// TIA Portal V17 export
// export: Created 2024-08-26T21:07:17.5555662Z, ExportSetting WithDefaults, DisplayName Totally Integrated Automation Portal, DisplayVersion V17 Update 7, DisplayName TIA Portal Openness, DisplayVersion V17 Update 7, DisplayName TIA Portal Version Control Interface, DisplayVersion V17, DisplayName SINAMICS Startdrive Advanced, DisplayVersion V17 SP2, DisplayName SINAMICS Startdrive G110M, G120, G120C, G120D, G120P, G115D, DisplayVersion V17 SP2, DisplayName SINAMICS Startdrive G130, G150, S120, S150, SINAMICS MV, S210, DisplayVersion V17 SP2, DisplayName STEP 7 Professional, DisplayVersion V17 Update 7, DisplayName STEP 7 Safety, DisplayVersion V17 Update 6, DisplayName WinCC Advanced / Unified PC, DisplayVersion V17 Update 7
DATA_BLOCK "CODE READING ANGLE"   // DB15
VERSION : 0.1
// stored: AutoNumber true, DBAccessibleFromOPCUA true, DBAccessibleFromWebserver true, InstanceOfName CODE READING, InstanceOfType FB
"CODE READING"
   // VAR_INPUT
   //    hwAdd : HW_IO := 385;
   //    scannerBusy : Bool := FALSE;
   //    autoMode : Bool := FALSE;
   //    manualMode : Bool := TRUE;
   //    scannerReadingComplete : Bool := FALSE;
   //    scannerReadingError : Bool := FALSE;
   //    clearData : Bool := FALSE;
   //    scannerDataSize : Int := 0;
   //    requestScannerAuto : Bool := FALSE;
   //    requestScannerManual : Bool := FALSE;
   //    scannerEnabled : Bool := TRUE;
   //    labelIdentyfier : String[5] := '06';
   //    labelPosition : Int := 4;
   //    labelIdentyfier_2 : String[5] := 'Y4';
   //    labelPosition_2 : Int := 5;
   //    label1 : Bool := TRUE;
   //    label2 : Bool := FALSE;
   // END_VAR
   // VAR_OUTPUT
   //    hmiLabel : String[180] := '';
   //    scannerOk : Bool := FALSE;
   //    scannerOk_2 : Bool := FALSE;
   //    clearReadComplete : Bool := FALSE;
   //    requestScannerOutput : Bool := FALSE;
   //    codeRead : Bool := FALSE;
   // END_VAR
   // VAR
   //    scannerReading { ExternalAccessible := 'False'; ExternalVisible := 'False'; ExternalWritable := 'False'} : Array[0..254] of Char;
   //    ScannerReadTimer { S7_SetPoint := 'True'} : TON_TIME;
   // END_VAR
BEGIN
   scannerReading[0] := '$00';
   scannerReading[1] := ',';
   scannerReading[2] := '$00';
   scannerReading[3] := ',';
   scannerReading[4] := '$00';
   scannerReading[5] := ',';
   scannerReading[6] := '$00';
   scannerReading[7] := '4';
   scannerReading[8] := '[';
   scannerReading[9] := ')';
   scannerReading[10] := '>';
   scannerReading[11] := '0';
   scannerReading[12] := '6';
   scannerReading[13] := 'P';
   scannerReading[14] := '1';
   scannerReading[15] := '3';
   scannerReading[16..17] := '5';
   scannerReading[18] := '1';
   scannerReading[19] := '8';
   scannerReading[20] := '0';
   scannerReading[21] := '4';
   scannerReading[22] := '1';
   scannerReading[23] := '2';
   scannerReading[24] := 'V';
   scannerReading[25] := '8';
   scannerReading[26] := '1';
   scannerReading[27] := '3';
   scannerReading[28] := '1';
   scannerReading[29] := '2';
   scannerReading[30] := '0';
   scannerReading[31] := '8';
   scannerReading[32] := '2';
   scannerReading[33] := '1';
   scannerReading[34] := 'T';
   scannerReading[35] := '2';
   scannerReading[36] := '4';
   scannerReading[37] := '1';
   scannerReading[38] := '2';
   scannerReading[39] := '9';
   scannerReading[40] := 'F';
   scannerReading[41] := '3';
   scannerReading[42] := '8';
   scannerReading[43] := '7';
   scannerReading[44] := '0';
   scannerReading[45] := '4';
   scannerReading[46] := '9';
   scannerReading[47] := '4';
   scannerReading[48] := '0';
   scannerReading[49] := '1';
   scannerReading[50..51] := 'I';
   scannerReading[52] := '4';
   scannerReading[53] := 'D';
   scannerReading[54] := '0';
   scannerReading[55] := '8';
   scannerReading[56] := '7';
   scannerReading[57] := 'X';
   scannerReading[58] := 'M';
   scannerReading[59] := '$R';
   scannerReading[60..135] := '$00';
   scannerReading[136..254] := ' ';
   ScannerReadTimer.PT := T#50MS;
   ScannerReadTimer.IN := FALSE;
END_DATA_BLOCK
